// TwinCAT 3 PLC project Device_Dummy
// ProgramVersion: 3.1.4023.0
// libraries:
//   Tc2_Standard, * (Beckhoff Automation GmbH)
//   Tc2_System, * (Beckhoff Automation GmbH)
//   Tc3_Module, * (Beckhoff Automation GmbH)
// project tree:
//   DUTs/ ST_StopStatus.TcDUT
//   / PlcTask.TcTTO
//   POUs/ MAIN.TcPOU, ReferenceBlock.TcPOU

CONFIGURATION Device_Dummy
    RESOURCE PLC ON TwinCAT3
        TASK PlcTask(INTERVAL := T#10ms, PRIORITY := 20);
        PROGRAM MAIN WITH PlcTask : MAIN;
    END_RESOURCE
END_CONFIGURATION

// ---- DUTs/ST_StopStatus.TcDUT
TYPE ST_StopStatus :
STRUCT
	PalletPresent :					BOOL;
	ReadyToAccept :					BOOL;
	PathClear :						BOOL;
	ToolingClear :					BOOL;
	InTransit :						BOOL;
END_STRUCT
END_TYPE

// ---- POUs/MAIN.TcPOU
PROGRAM MAIN
VAR_INPUT
	xInit			:BOOL:=TRUE;
END_VAR
VAR
	fbRef : ReferenceBlock;
END_VAR

IF xInit THEN
	xInit:=FALSE;
	fbRef();
END_IF

END_PROGRAM

// ---- POUs/ReferenceBlock.TcPOU
FUNCTION_BLOCK ReferenceBlock

VAR
	stStopStatus	:ST_StopStatus;
	refStopStatus	:REFERENCE TO ST_StopStatus;
END_VAR

refStopStatus REF= stStopStatus;

END_FUNCTION_BLOCK
